// TIA Portal V16 export
// export: Created 2022-11-24T15:20:55.0136242Z, ExportSetting WithDefaults, DisplayName Totally Integrated Automation Portal, DisplayVersion V16 Update 6, DisplayName TIA Portal Version Control Interface, DisplayVersion V16 Update 2, DisplayName TIA Portal Openness, DisplayVersion V16 Update 6, DisplayName SINAMICS Startdrive Advanced, DisplayVersion V16 Update 5, DisplayName SINAMICS Startdrive G130, G150, S120, S150, SINAMICS MV, S210, DisplayVersion V16 Update 5, DisplayName SINAMICS Startdrive G110M, G120, G120C, G120D, G120P, G115D, DisplayVersion V16 Update 5, DisplayName STEP 7 Professional, DisplayVersion V16 Update 6, DisplayName STEP 7 Safety, DisplayVersion V16, DisplayName WinCC Advanced, DisplayVersion V16 Update 6
FUNCTION "FC45_PrestretchPGSM_PGSA" : Void   // FC45, LAD
TITLE = Prestretch PGSM and PGSA management (HS30, Helix One)
{ S7_Optimized_Access := 'FALSE' }
AUTHOR : Robopac
VERSION : 0.0
// stored: AutoNumber false, IsIECCheckEnabled false, SetENOAutomatically false, UDAEnableTagReadback false
   VAR_TEMP
      TempInt : Int;
      TempDint : DInt;
      TempDint_2 : DInt;
      TiroStepTemp : Int;
      TiroFineTemp : Int;
   END_VAR
   VAR_TEMP   // added for the SCL form of the ladder/FBD networks
      _w1 : Bool;
      _w2 : Bool;
      _w3 : Bool;
      _w4 : Bool;
      _w5 : Bool;
      _w6 : Bool;
      _w7 : Bool;
   END_VAR
BEGIN

REGION Network 1: Film broken delay for spool carriage
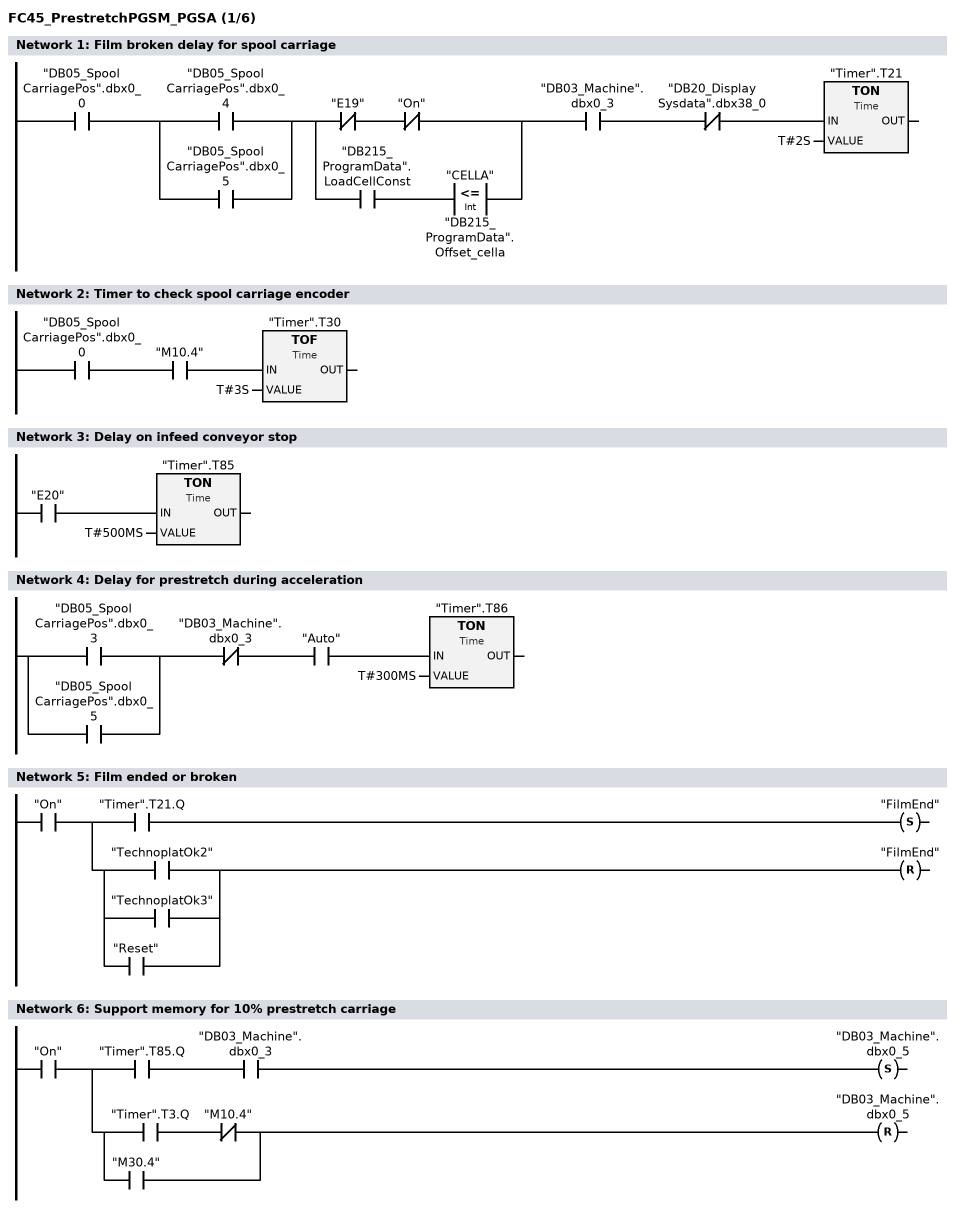
   "Timer".T21.TON(IN := "DB05_SpoolCarriagePos".dbx0_0 AND ("DB05_SpoolCarriagePos".dbx0_4 OR "DB05_SpoolCarriagePos".dbx0_5) AND ((NOT "E19" AND NOT "On") OR ("DB215_ProgramData".LoadCellConst AND ("CELLA" <= "DB215_ProgramData".Offset_cella))) AND "DB03_Machine".dbx0_3 AND NOT "DB20_DisplaySysdata".dbx38_0, PT := T#2S);   // TON coil
END_REGION

REGION Network 2: Timer to check spool carriage encoder
   "Timer".T30.TOF(IN := "DB05_SpoolCarriagePos".dbx0_0 AND "M10.4", PT := T#3S);   // TOF coil
END_REGION

REGION Network 3: Delay on infeed conveyor stop
   "Timer".T85.TON(IN := "E20", PT := T#500MS);   // TON coil
END_REGION

REGION Network 4: Delay for prestretch during acceleration
   "Timer".T86.TON(IN := ("DB05_SpoolCarriagePos".dbx0_3 OR "DB05_SpoolCarriagePos".dbx0_5) AND NOT "DB03_Machine".dbx0_3 AND "Auto", PT := T#300MS);   // TON coil
END_REGION

REGION Network 5: Film ended or broken
   RUNG wire#powerrail
      Contact( "On" )
      wire#w1
      Contact( "Timer".T21.Q )
      S_Coil( "FilmEnd" )
   END_RUNG
   RUNG wire#w1
      Contact( "TechnoplatOk2" )
      wire#w2
      R_Coil( "FilmEnd" )
   END_RUNG
   RUNG wire#w1
      Contact( "TechnoplatOk3" )
   END_RUNG wire#w2
   RUNG wire#w1
      Contact( "Reset" )
   END_RUNG wire#w2
   // the same network as SCL:
   IF "On" AND "Timer".T21.Q THEN "FilmEnd" := TRUE; END_IF;
   IF "On" AND ("TechnoplatOk2" OR "TechnoplatOk3" OR "Reset") THEN "FilmEnd" := FALSE; END_IF;
END_REGION

REGION Network 6: Support memory for 10% prestretch carriage
   RUNG wire#powerrail
      Contact( "On" )
      wire#w1
      Contact( "Timer".T85.Q )
      Contact( "DB03_Machine".dbx0_3 )
      S_Coil( "DB03_Machine".dbx0_5 )
   END_RUNG
   RUNG wire#w1
      Contact( "Timer".T3.Q )
      I_Contact( "M10.4" )
      wire#w2
      R_Coil( "DB03_Machine".dbx0_5 )
   END_RUNG
   RUNG wire#w1
      Contact( "M30.4" )
   END_RUNG wire#w2
   // the same network as SCL:
   IF "On" AND "Timer".T85.Q AND "DB03_Machine".dbx0_3 THEN "DB03_Machine".dbx0_5 := TRUE; END_IF;
   IF "On" AND (("Timer".T3.Q AND NOT "M10.4") OR "M30.4") THEN "DB03_Machine".dbx0_5 := FALSE; END_IF;
END_REGION

REGION Network 7: Support memory for prestretch PGSM or PGSA
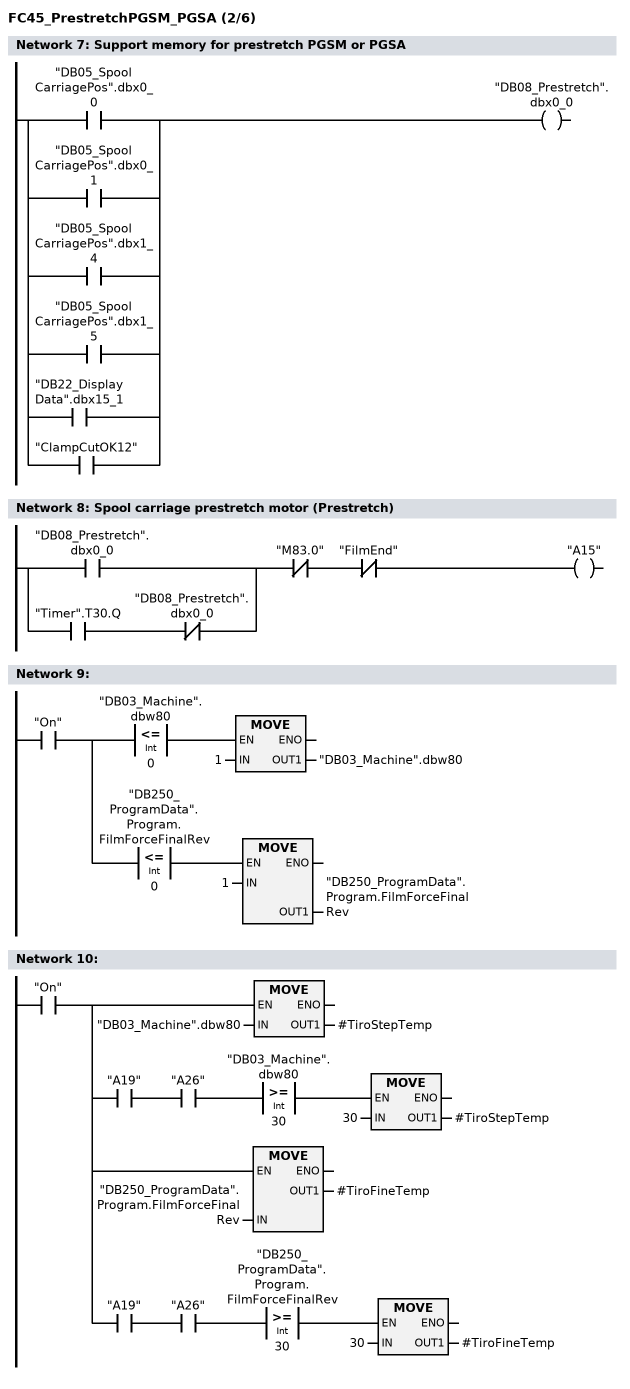
   RUNG wire#powerrail
      Contact( "DB05_SpoolCarriagePos".dbx0_0 )
      wire#w1
      Coil( "DB08_Prestretch".dbx0_0 )
   END_RUNG
   RUNG wire#powerrail
      Contact( "DB05_SpoolCarriagePos".dbx0_1 )
   END_RUNG wire#w1
   RUNG wire#powerrail
      Contact( "DB05_SpoolCarriagePos".dbx1_4 )
   END_RUNG wire#w1
   RUNG wire#powerrail
      Contact( "DB05_SpoolCarriagePos".dbx1_5 )
   END_RUNG wire#w1
   RUNG wire#powerrail
      Contact( "DB22_DisplayData".dbx15_1 )
   END_RUNG wire#w1
   RUNG wire#powerrail
      Contact( "ClampCutOK12" )
   END_RUNG wire#w1
   // the same network as SCL:
   "DB08_Prestretch".dbx0_0 := "DB05_SpoolCarriagePos".dbx0_0 OR "DB05_SpoolCarriagePos".dbx0_1 OR "DB05_SpoolCarriagePos".dbx1_4 OR "DB05_SpoolCarriagePos".dbx1_5 OR "DB22_DisplayData".dbx15_1 OR "ClampCutOK12";
END_REGION

REGION Network 8: Spool carriage prestretch motor (Prestretch)
   RUNG wire#powerrail
      Contact( "DB08_Prestretch".dbx0_0 )
      wire#w1
      I_Contact( "M83.0" )
      I_Contact( "FilmEnd" )
      Coil( "A15" )
   END_RUNG
   RUNG wire#powerrail
      Contact( "Timer".T30.Q )
      I_Contact( "DB08_Prestretch".dbx0_0 )
   END_RUNG wire#w1
   // the same network as SCL:
   "A15" := ("DB08_Prestretch".dbx0_0 OR ("Timer".T30.Q AND NOT "DB08_Prestretch".dbx0_0)) AND NOT "M83.0" AND NOT "FilmEnd";
END_REGION

REGION Network 9
   RUNG wire#powerrail
      Contact( "On" )
      wire#w1
      { S7_Templates := "SrcType := Int" } LE_Contact(in1 := "DB03_Machine".dbw80, in2 := 0)
      { S7_GenerateENO := "TRUE" } Move(in := 1, out1 => "DB03_Machine".dbw80)
   END_RUNG
   RUNG wire#w1
      { S7_Templates := "SrcType := Int" } LE_Contact(in1 := "DB250_ProgramData".Program.FilmForceFinalRev, in2 := 0)
      { S7_GenerateENO := "TRUE" } Move(in := 1, out1 => "DB250_ProgramData".Program.FilmForceFinalRev)
   END_RUNG
   // the same network as SCL:
   IF "On" AND ("DB03_Machine".dbw80 <= 0) THEN "DB03_Machine".dbw80 := 1; END_IF;
   IF "On" AND ("DB250_ProgramData".Program.FilmForceFinalRev <= 0) THEN
       "DB250_ProgramData".Program.FilmForceFinalRev := 1;
   END_IF;
END_REGION

REGION Network 10
   RUNG wire#powerrail
      Contact( "On" )
      wire#w1
      { S7_GenerateENO := "TRUE" } Move(in := "DB03_Machine".dbw80, out1 => #TiroStepTemp)
   END_RUNG
   RUNG wire#w1
      Contact( "A19" )
      Contact( "A26" )
      { S7_Templates := "SrcType := Int" } GE_Contact(in1 := "DB03_Machine".dbw80, in2 := 30)
      { S7_GenerateENO := "TRUE" } Move(in := 30, out1 => #TiroStepTemp)
   END_RUNG
   RUNG wire#w1
      { S7_GenerateENO := "TRUE" } Move(in := "DB250_ProgramData".Program.FilmForceFinalRev, out1 => #TiroFineTemp)
   END_RUNG
   RUNG wire#w1
      Contact( "A19" )
      Contact( "A26" )
      { S7_Templates := "SrcType := Int" } GE_Contact(in1 := "DB250_ProgramData".Program.FilmForceFinalRev, in2 := 30)
      { S7_GenerateENO := "TRUE" } Move(in := 30, out1 => #TiroFineTemp)
   END_RUNG
   // the same network as SCL:
   IF "On" THEN #TiroStepTemp := "DB03_Machine".dbw80; END_IF;
   IF "On" AND "A19" AND "A26" AND ("DB03_Machine".dbw80 >= 30) THEN #TiroStepTemp := 30; END_IF;
   IF "On" THEN #TiroFineTemp := "DB250_ProgramData".Program.FilmForceFinalRev; END_IF;
   IF "On" AND "A19" AND "A26" AND ("DB250_ProgramData".Program.FilmForceFinalRev >= 30) THEN
       #TiroFineTemp := 30;
   END_IF;
END_REGION

REGION Network 11
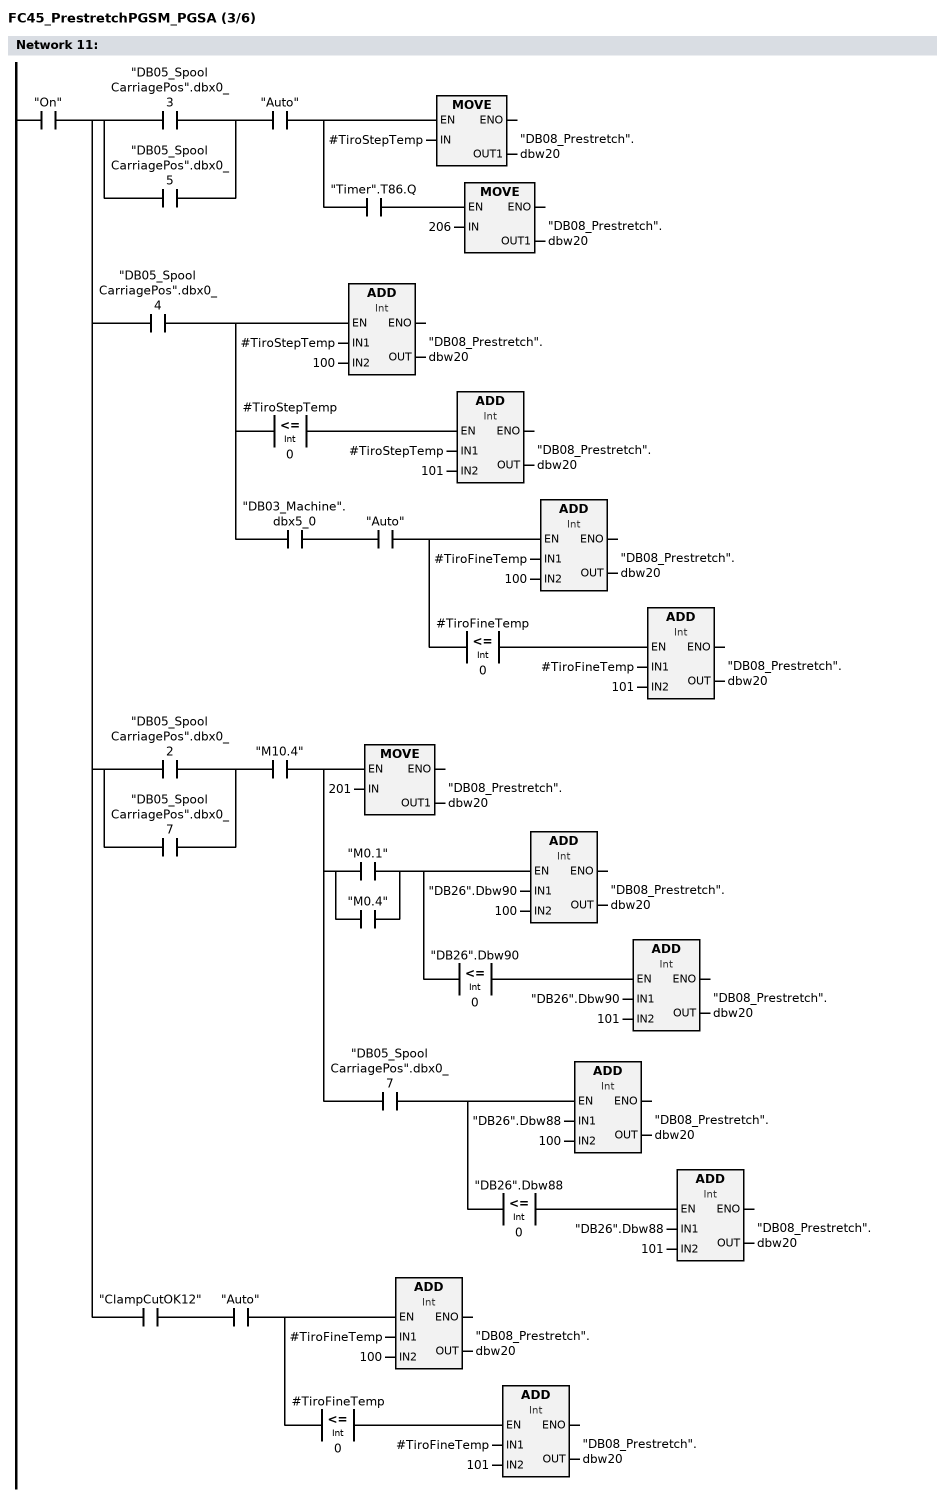
   RUNG wire#powerrail
      Contact( "On" )
      wire#w1
      Contact( "DB05_SpoolCarriagePos".dbx0_3 )
      wire#w2
      Contact( "Auto" )
      wire#w3
      { S7_GenerateENO := "TRUE" } Move(in := #TiroStepTemp, out1 => "DB08_Prestretch".dbw20)
   END_RUNG
   RUNG wire#w1
      Contact( "DB05_SpoolCarriagePos".dbx0_5 )
   END_RUNG wire#w2
   RUNG wire#w3
      Contact( "Timer".T86.Q )
      { S7_GenerateENO := "TRUE" } Move(in := 206, out1 => "DB08_Prestretch".dbw20)
   END_RUNG
   RUNG wire#w1
      Contact( "DB05_SpoolCarriagePos".dbx0_4 )
      wire#w4
      { S7_Templates := "SrcType := Int"; S7_GenerateENO := "TRUE" } Add(in1 := #TiroStepTemp, in2 := 100, out => "DB08_Prestretch".dbw20)
   END_RUNG
   RUNG wire#w4
      { S7_Templates := "SrcType := Int" } LE_Contact(in1 := #TiroStepTemp, in2 := 0)
      { S7_Templates := "SrcType := Int"; S7_GenerateENO := "TRUE" } Add(in1 := #TiroStepTemp, in2 := 101, out => "DB08_Prestretch".dbw20)
   END_RUNG
   RUNG wire#w4
      Contact( "DB03_Machine".dbx5_0 )
      Contact( "Auto" )
      wire#w5
      { S7_Templates := "SrcType := Int"; S7_GenerateENO := "TRUE" } Add(in1 := #TiroFineTemp, in2 := 100, out => "DB08_Prestretch".dbw20)
   END_RUNG
   RUNG wire#w5
      { S7_Templates := "SrcType := Int" } LE_Contact(in1 := #TiroFineTemp, in2 := 0)
      { S7_Templates := "SrcType := Int"; S7_GenerateENO := "TRUE" } Add(in1 := #TiroFineTemp, in2 := 101, out => "DB08_Prestretch".dbw20)
   END_RUNG
   RUNG wire#w1
      Contact( "DB05_SpoolCarriagePos".dbx0_2 )
      wire#w6
      Contact( "M10.4" )
      wire#w7
      { S7_GenerateENO := "TRUE" } Move(in := 201, out1 => "DB08_Prestretch".dbw20)
   END_RUNG
   RUNG wire#w1
      Contact( "DB05_SpoolCarriagePos".dbx0_7 )
   END_RUNG wire#w6
   RUNG wire#w7
      Contact( "M0.1" )
      wire#w8
      { S7_Templates := "SrcType := Int"; S7_GenerateENO := "TRUE" } Add(in1 := "DB26".Dbw90, in2 := 100, out => "DB08_Prestretch".dbw20)
   END_RUNG
   RUNG wire#w7
      Contact( "M0.4" )
   END_RUNG wire#w8
   RUNG wire#w8
      { S7_Templates := "SrcType := Int" } LE_Contact(in1 := "DB26".Dbw90, in2 := 0)
      { S7_Templates := "SrcType := Int"; S7_GenerateENO := "TRUE" } Add(in1 := "DB26".Dbw90, in2 := 101, out => "DB08_Prestretch".dbw20)
   END_RUNG
   RUNG wire#w7
      Contact( "DB05_SpoolCarriagePos".dbx0_7 )
      wire#w9
      { S7_Templates := "SrcType := Int"; S7_GenerateENO := "TRUE" } Add(in1 := "DB26".Dbw88, in2 := 100, out => "DB08_Prestretch".dbw20)
   END_RUNG
   RUNG wire#w9
      { S7_Templates := "SrcType := Int" } LE_Contact(in1 := "DB26".Dbw88, in2 := 0)
      { S7_Templates := "SrcType := Int"; S7_GenerateENO := "TRUE" } Add(in1 := "DB26".Dbw88, in2 := 101, out => "DB08_Prestretch".dbw20)
   END_RUNG
   RUNG wire#w1
      Contact( "ClampCutOK12" )
      Contact( "Auto" )
      wire#w10
      { S7_Templates := "SrcType := Int"; S7_GenerateENO := "TRUE" } Add(in1 := #TiroFineTemp, in2 := 100, out => "DB08_Prestretch".dbw20)
   END_RUNG
   RUNG wire#w10
      { S7_Templates := "SrcType := Int" } LE_Contact(in1 := #TiroFineTemp, in2 := 0)
      { S7_Templates := "SrcType := Int"; S7_GenerateENO := "TRUE" } Add(in1 := #TiroFineTemp, in2 := 101, out => "DB08_Prestretch".dbw20)
   END_RUNG
   // the same network as SCL:
   #_w1 := "On" AND ("DB05_SpoolCarriagePos".dbx0_3 OR "DB05_SpoolCarriagePos".dbx0_5) AND "Auto";
   IF #_w1 THEN "DB08_Prestretch".dbw20 := #TiroStepTemp; END_IF;
   IF #_w1 AND "Timer".T86.Q THEN "DB08_Prestretch".dbw20 := 206; END_IF;
   #_w2 := "On" AND "DB05_SpoolCarriagePos".dbx0_4;
   IF #_w2 THEN "DB08_Prestretch".dbw20 := #TiroStepTemp + 100; END_IF;
   IF #_w2 AND (#TiroStepTemp <= 0) THEN "DB08_Prestretch".dbw20 := #TiroStepTemp + 101; END_IF;
   #_w3 := #_w2 AND "DB03_Machine".dbx5_0 AND "Auto";
   IF #_w3 THEN "DB08_Prestretch".dbw20 := #TiroFineTemp + 100; END_IF;
   IF #_w3 AND (#TiroFineTemp <= 0) THEN "DB08_Prestretch".dbw20 := #TiroFineTemp + 101; END_IF;
   #_w4 := "On" AND ("DB05_SpoolCarriagePos".dbx0_2 OR "DB05_SpoolCarriagePos".dbx0_7) AND "M10.4";
   IF #_w4 THEN "DB08_Prestretch".dbw20 := 201; END_IF;
   #_w5 := #_w4 AND ("M0.1" OR "M0.4");
   IF #_w5 THEN "DB08_Prestretch".dbw20 := "DB26".Dbw90 + 100; END_IF;
   IF #_w5 AND ("DB26".Dbw90 <= 0) THEN "DB08_Prestretch".dbw20 := "DB26".Dbw90 + 101; END_IF;
   #_w6 := #_w4 AND "DB05_SpoolCarriagePos".dbx0_7;
   IF #_w6 THEN "DB08_Prestretch".dbw20 := "DB26".Dbw88 + 100; END_IF;
   IF #_w6 AND ("DB26".Dbw88 <= 0) THEN "DB08_Prestretch".dbw20 := "DB26".Dbw88 + 101; END_IF;
   #_w7 := "On" AND "ClampCutOK12" AND "Auto";
   IF #_w7 THEN "DB08_Prestretch".dbw20 := #TiroFineTemp + 100; END_IF;
   IF #_w7 AND (#TiroFineTemp <= 0) THEN "DB08_Prestretch".dbw20 := #TiroFineTemp + 101; END_IF;
END_REGION

REGION Network 12
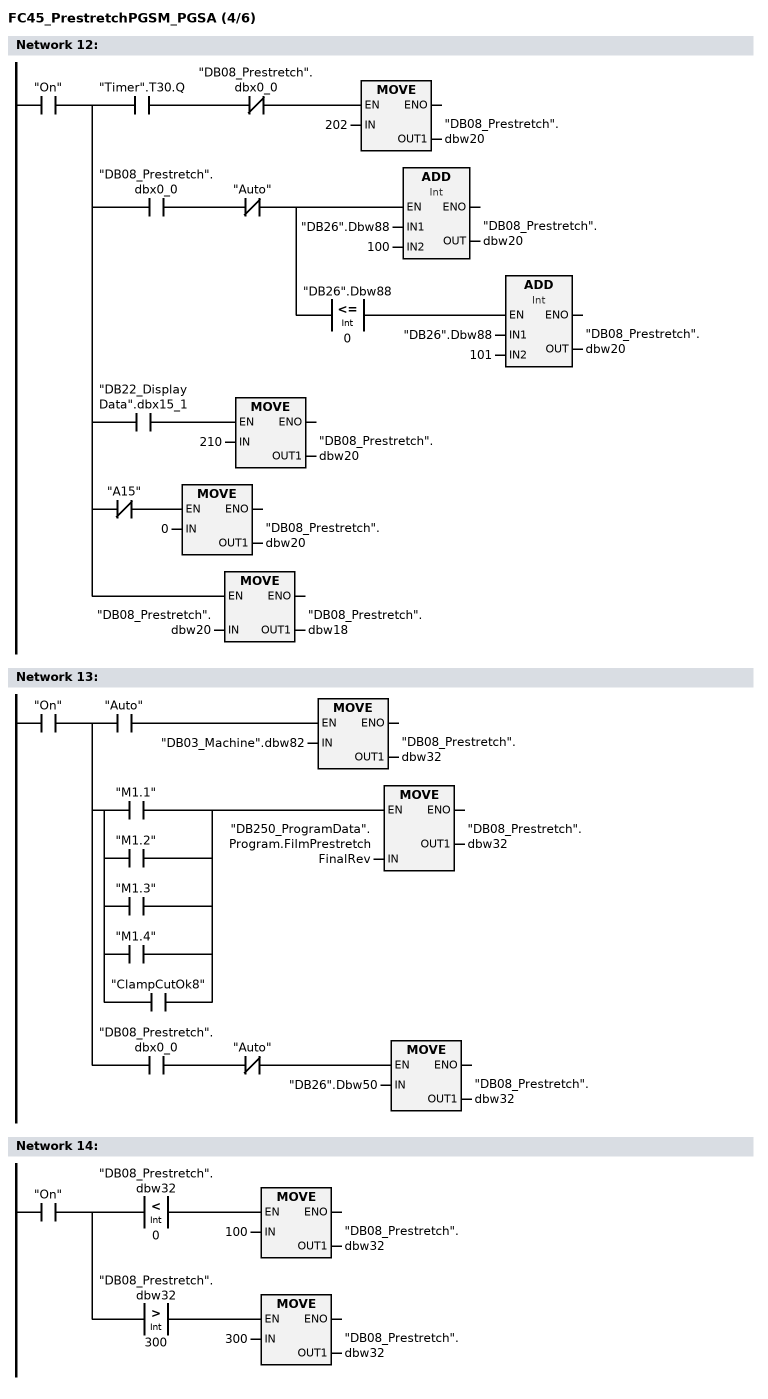
   RUNG wire#powerrail
      Contact( "On" )
      wire#w1
      Contact( "Timer".T30.Q )
      I_Contact( "DB08_Prestretch".dbx0_0 )
      { S7_GenerateENO := "TRUE" } Move(in := 202, out1 => "DB08_Prestretch".dbw20)
   END_RUNG
   RUNG wire#w1
      Contact( "DB08_Prestretch".dbx0_0 )
      I_Contact( "Auto" )
      wire#w2
      { S7_Templates := "SrcType := Int"; S7_GenerateENO := "TRUE" } Add(in1 := "DB26".Dbw88, in2 := 100, out => "DB08_Prestretch".dbw20)
   END_RUNG
   RUNG wire#w2
      { S7_Templates := "SrcType := Int" } LE_Contact(in1 := "DB26".Dbw88, in2 := 0)
      { S7_Templates := "SrcType := Int"; S7_GenerateENO := "TRUE" } Add(in1 := "DB26".Dbw88, in2 := 101, out => "DB08_Prestretch".dbw20)
   END_RUNG
   RUNG wire#w1
      Contact( "DB22_DisplayData".dbx15_1 )
      { S7_GenerateENO := "TRUE" } Move(in := 210, out1 => "DB08_Prestretch".dbw20)
   END_RUNG
   RUNG wire#w1
      I_Contact( "A15" )
      { S7_GenerateENO := "TRUE" } Move(in := 0, out1 => "DB08_Prestretch".dbw20)
   END_RUNG
   RUNG wire#w1
      { S7_GenerateENO := "TRUE" } Move(in := "DB08_Prestretch".dbw20, out1 => "DB08_Prestretch".dbw18)
   END_RUNG
   // the same network as SCL:
   IF "On" AND "Timer".T30.Q AND NOT "DB08_Prestretch".dbx0_0 THEN "DB08_Prestretch".dbw20 := 202; END_IF;
   #_w1 := "On" AND "DB08_Prestretch".dbx0_0 AND NOT "Auto";
   IF #_w1 THEN "DB08_Prestretch".dbw20 := "DB26".Dbw88 + 100; END_IF;
   IF #_w1 AND ("DB26".Dbw88 <= 0) THEN "DB08_Prestretch".dbw20 := "DB26".Dbw88 + 101; END_IF;
   IF "On" AND "DB22_DisplayData".dbx15_1 THEN "DB08_Prestretch".dbw20 := 210; END_IF;
   IF "On" AND NOT "A15" THEN "DB08_Prestretch".dbw20 := 0; END_IF;
   IF "On" THEN "DB08_Prestretch".dbw18 := "DB08_Prestretch".dbw20; END_IF;
END_REGION

REGION Network 13
   RUNG wire#powerrail
      Contact( "On" )
      wire#w1
      Contact( "Auto" )
      { S7_GenerateENO := "TRUE" } Move(in := "DB03_Machine".dbw82, out1 => "DB08_Prestretch".dbw32)
   END_RUNG
   RUNG wire#w1
      Contact( "M1.1" )
      wire#w2
      { S7_GenerateENO := "TRUE" } Move(in := "DB250_ProgramData".Program.FilmPrestretchFinalRev, out1 => "DB08_Prestretch".dbw32)
   END_RUNG
   RUNG wire#w1
      Contact( "M1.2" )
   END_RUNG wire#w2
   RUNG wire#w1
      Contact( "M1.3" )
   END_RUNG wire#w2
   RUNG wire#w1
      Contact( "M1.4" )
   END_RUNG wire#w2
   RUNG wire#w1
      Contact( "ClampCutOk8" )
   END_RUNG wire#w2
   RUNG wire#w1
      Contact( "DB08_Prestretch".dbx0_0 )
      I_Contact( "Auto" )
      { S7_GenerateENO := "TRUE" } Move(in := "DB26".Dbw50, out1 => "DB08_Prestretch".dbw32)
   END_RUNG
   // the same network as SCL:
   IF "On" AND "Auto" THEN "DB08_Prestretch".dbw32 := "DB03_Machine".dbw82; END_IF;
   IF "On" AND ("M1.1" OR "M1.2" OR "M1.3" OR "M1.4" OR "ClampCutOk8") THEN
       "DB08_Prestretch".dbw32 := "DB250_ProgramData".Program.FilmPrestretchFinalRev;
   END_IF;
   IF "On" AND "DB08_Prestretch".dbx0_0 AND NOT "Auto" THEN "DB08_Prestretch".dbw32 := "DB26".Dbw50; END_IF;
END_REGION

REGION Network 14
   RUNG wire#powerrail
      Contact( "On" )
      wire#w1
      { S7_Templates := "SrcType := Int" } LT_Contact(in1 := "DB08_Prestretch".dbw32, in2 := 0)
      { S7_GenerateENO := "TRUE" } Move(in := 100, out1 => "DB08_Prestretch".dbw32)
   END_RUNG
   RUNG wire#w1
      { S7_Templates := "SrcType := Int" } GT_Contact(in1 := "DB08_Prestretch".dbw32, in2 := 300)
      { S7_GenerateENO := "TRUE" } Move(in := 300, out1 => "DB08_Prestretch".dbw32)
   END_RUNG
   // the same network as SCL:
   IF "On" AND ("DB08_Prestretch".dbw32 < 0) THEN "DB08_Prestretch".dbw32 := 100; END_IF;
   IF "On" AND ("DB08_Prestretch".dbw32 > 300) THEN "DB08_Prestretch".dbw32 := 300; END_IF;
END_REGION

REGION Network 15
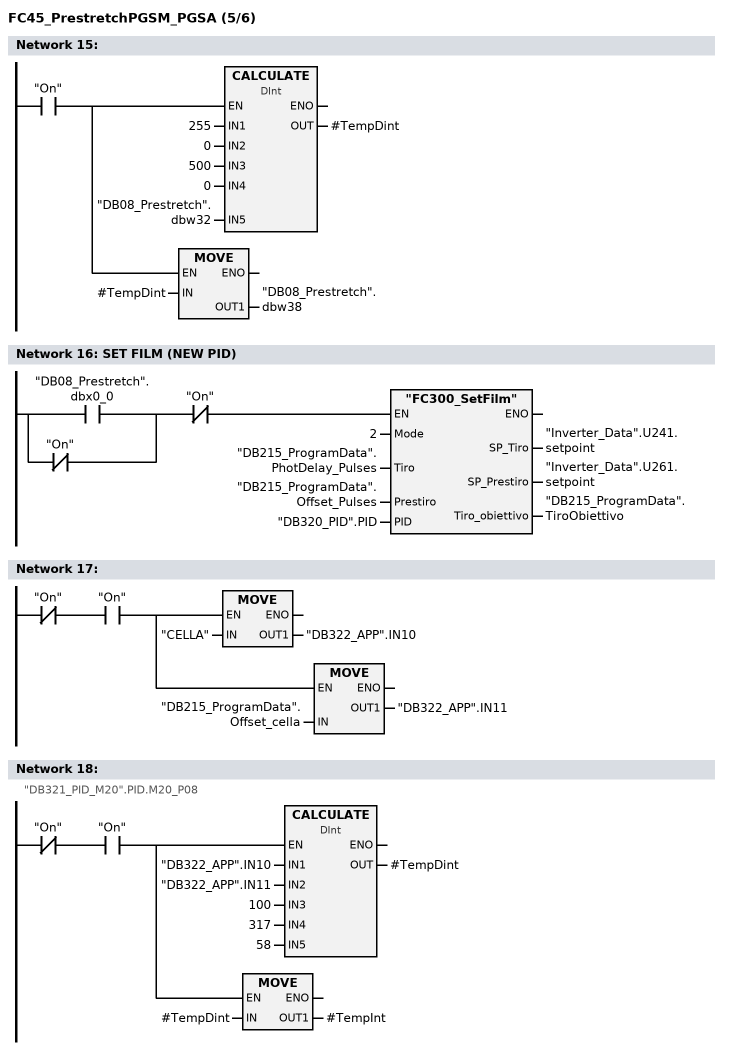
   RUNG wire#powerrail
      Contact( "On" )
      wire#w1
      { S7_Templates := "SrcType := DInt"; S7_GenerateENO := "TRUE"; S7_Expression := "((IN5-IN4)*(IN1-IN2)/(IN3-IN4))+IN2" } Calculate(in1 := 255, in2 := 0, in3 := 500, in4 := 0, in5 := "DB08_Prestretch".dbw32, out => #TempDint)
   END_RUNG
   RUNG wire#w1
      { S7_GenerateENO := "TRUE" } Move(in := #TempDint, out1 => "DB08_Prestretch".dbw38)
   END_RUNG
   // the same network as SCL:
   IF "On" THEN
       #TempDint := (("DB08_Prestretch".dbw32-0)*(255-0)/(500-0))+0;
       "DB08_Prestretch".dbw38 := #TempDint;
   END_IF;
END_REGION

REGION Network 16: SET FILM (NEW PID)
   RUNG wire#powerrail
      Contact( "DB08_Prestretch".dbx0_0 )
      wire#w1
      I_Contact( "On" )
      "FC300_SetFilm"(Mode := 2, Tiro := "DB215_ProgramData".PhotDelay_Pulses, Prestiro := "DB215_ProgramData".Offset_Pulses, PID := "DB320_PID".PID, SP_Tiro => "Inverter_Data".U241.setpoint, SP_Prestiro => "Inverter_Data".U261.setpoint, Tiro_obiettivo => "DB215_ProgramData".TiroObiettivo)
   END_RUNG
   RUNG wire#powerrail
      I_Contact( "On" )
   END_RUNG wire#w1
   // the same network as SCL:
   IF ("DB08_Prestretch".dbx0_0 OR NOT "On") AND NOT "On" THEN
       "FC300_SetFilm"(Mode := 2,
                       Tiro := "DB215_ProgramData".PhotDelay_Pulses,
                       Prestiro := "DB215_ProgramData".Offset_Pulses,
                       PID := "DB320_PID".PID,
                       SP_Tiro => "Inverter_Data".U241.setpoint,
                       SP_Prestiro => "Inverter_Data".U261.setpoint,
                       Tiro_obiettivo => "DB215_ProgramData".TiroObiettivo);
   END_IF;
END_REGION

REGION Network 17
   RUNG wire#powerrail
      I_Contact( "On" )
      Contact( "On" )
      wire#w1
      Move(in := "CELLA", out1 => "DB322_APP".IN10)
   END_RUNG
   RUNG wire#w1
      Move(in := "DB215_ProgramData".Offset_cella, out1 => "DB322_APP".IN11)
   END_RUNG
   // the same network as SCL:
   IF NOT "On" AND "On" THEN
       "DB322_APP".IN10 := "CELLA";
       "DB322_APP".IN11 := "DB215_ProgramData".Offset_cella;
   END_IF;
END_REGION

REGION Network 18
   // "DB321_PID_M20".PID.M20_P08
   RUNG wire#powerrail
      I_Contact( "On" )
      Contact( "On" )
      wire#w1
      { S7_Templates := "SrcType := DInt"; S7_Expression := "((IN1-IN2)*IN3/IN4)+IN5" } Calculate(in1 := "DB322_APP".IN10, in2 := "DB322_APP".IN11, in3 := 100, in4 := 317, in5 := 58, out => #TempDint)
   END_RUNG
   RUNG wire#w1
      Move(in := #TempDint, out1 => #TempInt)
   END_RUNG
   // the same network as SCL:
   IF NOT "On" AND "On" THEN
       #TempDint := (("DB322_APP".IN10-"DB322_APP".IN11)*100/317)+58;
       #TempInt := #TempDint;
   END_IF;
END_REGION

REGION Network 19
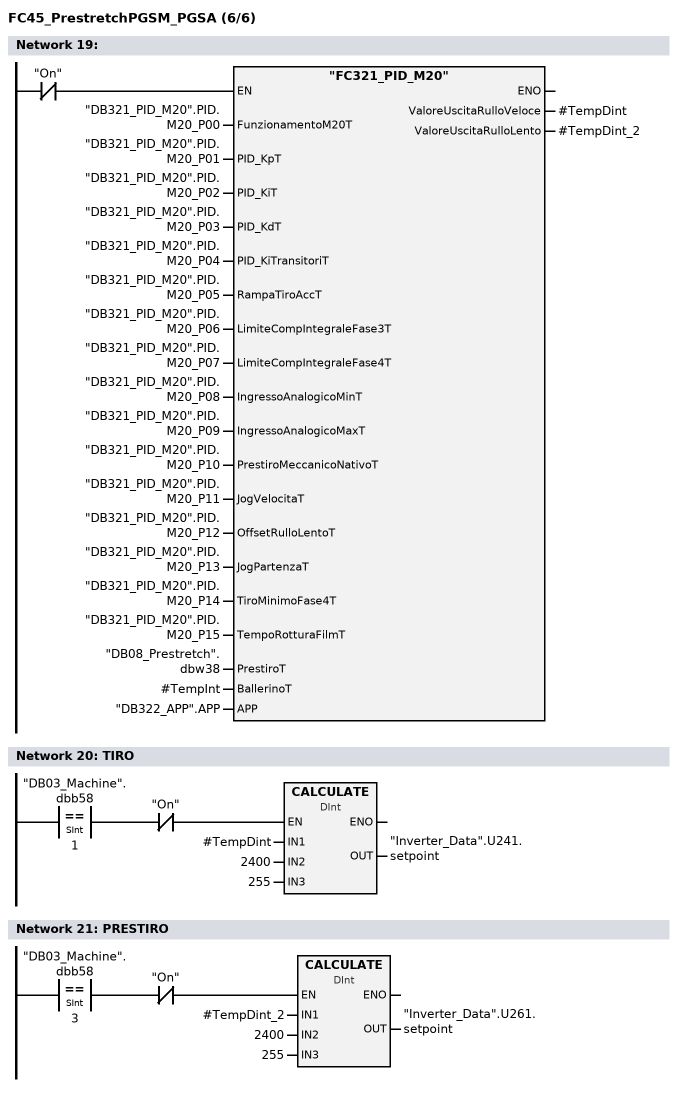
   RUNG wire#powerrail
      I_Contact( "On" )
      "FC321_PID_M20"(FunzionamentoM20T := "DB321_PID_M20".PID.M20_P00, PID_KpT := "DB321_PID_M20".PID.M20_P01, PID_KiT := "DB321_PID_M20".PID.M20_P02, PID_KdT := "DB321_PID_M20".PID.M20_P03, PID_KiTransitoriT := "DB321_PID_M20".PID.M20_P04, RampaTiroAccT := "DB321_PID_M20".PID.M20_P05, LimiteCompIntegraleFase3T := "DB321_PID_M20".PID.M20_P06, LimiteCompIntegraleFase4T := "DB321_PID_M20".PID.M20_P07, IngressoAnalogicoMinT := "DB321_PID_M20".PID.M20_P08, IngressoAnalogicoMaxT := "DB321_PID_M20".PID.M20_P09, PrestiroMeccanicoNativoT := "DB321_PID_M20".PID.M20_P10, JogVelocitaT := "DB321_PID_M20".PID.M20_P11, OffsetRulloLentoT := "DB321_PID_M20".PID.M20_P12, JogPartenzaT := "DB321_PID_M20".PID.M20_P13, TiroMinimoFase4T := "DB321_PID_M20".PID.M20_P14, TempoRotturaFilmT := "DB321_PID_M20".PID.M20_P15, PrestiroT := "DB08_Prestretch".dbw38, BallerinoT := #TempInt, APP := "DB322_APP".APP, ValoreUscitaRulloVeloce => #TempDint, ValoreUscitaRulloLento => #TempDint_2)
   END_RUNG
   // the same network as SCL:
   IF NOT "On" THEN
       "FC321_PID_M20"(FunzionamentoM20T := "DB321_PID_M20".PID.M20_P00,
                       PID_KpT := "DB321_PID_M20".PID.M20_P01,
                       PID_KiT := "DB321_PID_M20".PID.M20_P02,
                       PID_KdT := "DB321_PID_M20".PID.M20_P03,
                       PID_KiTransitoriT := "DB321_PID_M20".PID.M20_P04,
                       RampaTiroAccT := "DB321_PID_M20".PID.M20_P05,
                       LimiteCompIntegraleFase3T := "DB321_PID_M20".PID.M20_P06,
                       LimiteCompIntegraleFase4T := "DB321_PID_M20".PID.M20_P07,
                       IngressoAnalogicoMinT := "DB321_PID_M20".PID.M20_P08,
                       IngressoAnalogicoMaxT := "DB321_PID_M20".PID.M20_P09,
                       PrestiroMeccanicoNativoT := "DB321_PID_M20".PID.M20_P10,
                       JogVelocitaT := "DB321_PID_M20".PID.M20_P11,
                       OffsetRulloLentoT := "DB321_PID_M20".PID.M20_P12,
                       JogPartenzaT := "DB321_PID_M20".PID.M20_P13,
                       TiroMinimoFase4T := "DB321_PID_M20".PID.M20_P14,
                       TempoRotturaFilmT := "DB321_PID_M20".PID.M20_P15,
                       PrestiroT := "DB08_Prestretch".dbw38,
                       BallerinoT := #TempInt,
                       APP := "DB322_APP".APP,
                       ValoreUscitaRulloVeloce => #TempDint,
                       ValoreUscitaRulloLento => #TempDint_2);
   END_IF;
END_REGION

REGION Network 20: TIRO
   RUNG wire#powerrail
      { S7_Templates := "SrcType := SInt" } EQ_Contact(in1 := "DB03_Machine".dbb58, in2 := 1)
      I_Contact( "On" )
      { S7_Templates := "SrcType := DInt"; S7_Expression := "IN1*IN2/IN3" } Calculate(in1 := #TempDint, in2 := 2400, in3 := 255, out => "Inverter_Data".U241.setpoint)
   END_RUNG
   // the same network as SCL:
   IF ("DB03_Machine".dbb58 = 1) AND NOT "On" THEN
       "Inverter_Data".U241.setpoint := #TempDint*2400/255;
   END_IF;
END_REGION

REGION Network 21: PRESTIRO
   RUNG wire#powerrail
      { S7_Templates := "SrcType := SInt" } EQ_Contact(in1 := "DB03_Machine".dbb58, in2 := 3)
      I_Contact( "On" )
      { S7_Templates := "SrcType := DInt"; S7_Expression := "IN1*IN2/IN3" } Calculate(in1 := #TempDint_2, in2 := 2400, in3 := 255, out => "Inverter_Data".U261.setpoint)
   END_RUNG
   // the same network as SCL:
   IF ("DB03_Machine".dbb58 = 3) AND NOT "On" THEN
       "Inverter_Data".U261.setpoint := #TempDint_2*2400/255;
   END_IF;
END_REGION
END_FUNCTION
